KUKA KRL program: chk_w1_wechs_ok.src

&ACCESS RVO5
&REL 16
&COMMENT Check c1
DEF chk_w1_wechs_ok( )
;Diag_Appl(#on,5)

; VERIFICAÇÃO DE FERRAMENTA: C1

$TIMER[10] = 0
$TIMER_STOP[10] = FALSE

wait for ((not  $in[161]) and (($in[169]) or (NOT( $in[169]) and $in[3320])) and ($in [177]) and ($in [185]) and ( $in[219]))



$TIMER_STOP[10] = TRUE
$TIMER[10] = 0

;//---- End -------
;Diag_Appl(#Off,5)
END
